PROGRAM MAIN
VAR

END_VAR

// Call Connection Program for Connection with Factory IO Modbus Server //
Connection();
// Call Demo Program
DemoProgram();

END_PROGRAM

(* stored: Version 1.1.0.1
   POU MAIN: Id {e8fbe9ec-1542-41ae-b58e-a7b3e7e6778f}, SpecialFunc None *)
